PROGRAM MAIN
VAR
	fbMachine : Machine;
	State : INT := 0;
	Reset : BOOL;
	Start : BOOL;
	Clear : BOOL;
	Abort : BOOL;
END_VAR

CASE State OF
	0:
		IF fbMachine.Initialise() THEN
			State := 1;
		END_IF
	1:
		fbMachine.Cycle();
END_CASE

IF Reset THEN
	fbMachine.SetPackML(state := E_PMLCommand.ePMLCommand_Reset);
	Reset := FALSE;
END_IF
IF Abort THEN
	fbMachine.SetPackML(state := E_PMLCommand.ePMLCommand_Abort);
	Abort := FALSE;
END_IF
IF Clear THEN
	fbMachine.SetPackML(state := E_PMLCommand.ePMLCommand_Clear);
	Clear := FALSE;
END_IF
IF Start THEN
	fbMachine.SetPackML(state := E_PMLCommand.ePMLCommand_Start);
	Start := FALSE;
END_IF

result := foo.METH();

END_PROGRAM

(* stored: Version 1.1.0.1, ProductVersion 3.1.4024.12
   POU MAIN: Id {c3798e48-78cc-4657-a79b-2d5c7d932da8}, SpecialFunc None *)
